// TIA Portal V20 export
TYPE "LKinCtrl_PathEditor_typeCommandEditorInternalEvents"
// stored: Access Published
   STRUCT
      openLinkTable { ExternalAccessible := 'False'; ExternalVisible := 'False'; ExternalWritable := 'False'} : Bool;
      openCommandEditor { ExternalAccessible := 'False'; ExternalVisible := 'False'; ExternalWritable := 'False'} : Bool;
      closeCommandEditor { ExternalAccessible := 'False'; ExternalVisible := 'False'; ExternalWritable := 'False'} : Bool;
      selectionChanged { ExternalAccessible := 'False'; ExternalVisible := 'False'; ExternalWritable := 'False'} : Struct
         trigger : Bool;   // triggers internal event. Reset internally.
         selectedIndex : DInt;   // 10: variables, 11: conditions, 12: Inputs, 13: Outputs, 14: Points, 20: Axes, 21: PosSyncAxes , 22: SyncAxes, 30: Labels, 40: Sequences
         noSelection : Bool;
         contentType : Int;   // show only used values.
      END_STRUCT;
      commandSelectionChanged { ExternalAccessible := 'False'; ExternalVisible := 'False'; ExternalWritable := 'False'} : Struct
         trigger : Bool;
         mode : USInt;   // 0: add, 1: edit
         command : "LKinCtrl_typePathDataElement";
      END_STRUCT;
   END_STRUCT;
END_TYPE
